DATA_BLOCK "KukaRobot1_CtrlDB"
{ S7_Optimized_Access := 'FALSE' }
VERSION : 0.1
"KukaRobot1_Ctrl"

BEGIN

END_DATA_BLOCK

